FUNCTION_BLOCK I_WBSD (* Service Interface Function Block Type *)
  (* Standard: ISO 11783-7; Classification: PGN 65096; Function: Wheel-based Speed and Distance WBSD; Description: Message sent by the Tractor ECU on the implement bus on construction and agricultural implements providing to connected systems the current measured wheel-based speed. The message also includes a free-running distance counter, an indication of the direction of travel and the state of the start/stop switch or input. When the ignition key switch is turned off, both the ECU_PWR and PWR have to be maintained to send this message for an additional 2 s. This is not required when the engine is cranking (starting). Accuracies of both wheel-based and ground-based sources can be speed-dependent and degrade at low speeds. Wheel-based information might not be updated at the 100 ms rate at low speeds. https://www.isobus.net/isobus/pGNAndSPN/14648?type=PGN *)
  (* Version 1.0, 2024-07-09, franz *)
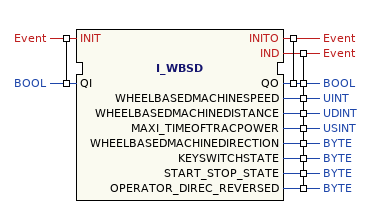
  EVENT_INPUT
    INIT WITH QI; (* Service Initialization *)
  END_EVENT
  EVENT_OUTPUT
    INITO WITH QO; (* Initialization Confirm *)
    IND WITH QO, WHEELBASEDMACHINESPEED, WHEELBASEDMACHINEDISTANCE, MAXI_TIMEOFTRACPOWER, WHEELBASEDMACHINEDIRECTION, KEYSWITCHSTATE, START_STOP_STATE, OPERATOR_DIREC_REVERSED; (* Indication from Resource *)
  END_EVENT
  VAR_INPUT
    QI : BOOL; (* Event Input Qualifier *)
  END_VAR
  VAR_OUTPUT
    QO : BOOL; (* Event Output Qualifier *)
    WHEELBASEDMACHINESPEED : UINT; (* Wheel-based machine speed *)
    WHEELBASEDMACHINEDISTANCE : UDINT; (* Wheel-based machine distance *)
    MAXI_TIMEOFTRACPOWER : USINT; (* Maximum Time of Tractor Power *)
    WHEELBASEDMACHINEDIRECTION : BYTE; (* Wheel-based machine direction *)
    KEYSWITCHSTATE : BYTE; (* Key switch state *)
    START_STOP_STATE : BYTE; (* Implement Start/Stop operations *)
    OPERATOR_DIREC_REVERSED : BYTE; (* Operator direction reversed *)
  END_VAR
  SERVICE APPLICATION/RESOURCE (* Service Interface Function Block Type *)
    SEQUENCE normal_establishment
      APPLICATION.INIT+(PARAMS) -> RESOURCE.initialize(PARAMS) -> APPLICATION.INITO+();
    END_SEQUENCE
    SEQUENCE unsuccessful_establishment
      APPLICATION.INIT+(PARAMS) -> RESOURCE.initialize(PARAMS) -> APPLICATION.INITO-(STATUS);
    END_SEQUENCE
    SEQUENCE request_confirm
      APPLICATION.REQ+(SD) -> RESOURCE.request(SD) -> APPLICATION.CNF+(RD);
    END_SEQUENCE
    SEQUENCE request_inhibited
      APPLICATION.REQ-(SD) -> APPLICATION.CNF-(STATUS);
    END_SEQUENCE
    SEQUENCE request_error
      APPLICATION.REQ+(SD) -> RESOURCE.request(SD) -> APPLICATION.CNF-(STATUS);
    END_SEQUENCE
    SEQUENCE indication_response
      RESOURCE.indicate(RD) -> APPLICATION.IND+(RD);
      APPLICATION.RSP(QI,SD) -> RESOURCE.response(QI,SD);
    END_SEQUENCE
    SEQUENCE indication_inhibited
      RESOURCE.indicate(RD,QI=FALSE) -> RESOURCE.inhibited();
    END_SEQUENCE
    SEQUENCE error_indication
      RESOURCE.error(STATUS) -> APPLICATION.IND-(STATUS);
    END_SEQUENCE
    SEQUENCE application_initiated_termination
      APPLICATION.INIT-() -> RESOURCE.terminate() -> APPLICATION.INITO-(STATUS);
    END_SEQUENCE
    SEQUENCE resource_initiated_termination
      -> APPLICATION.INITO-(STATUS);
    END_SEQUENCE
  END_SERVICE
END_FUNCTION_BLOCK
